INTERFACE I_InterfaceDatatype EXTENDS I_Datatype

PROPERTY PUBLIC Identifier : T_MAXSTRING
GET
END_GET
END_PROPERTY

END_INTERFACE

(* stored: Version 1.1.0.1, ProductVersion 3.1.4024.12
   Itf I_InterfaceDatatype: Id {323088ec-6ba5-4fe0-afdb-47275dc98016}
   Property Identifier: Id {6c55f951-bca8-4037-92fa-277b77548ef1}
   Get Get: Id {a8ca722f-9607-4d3f-8b6a-5cf70a3d9178} *)
